Staubli VAL3: movToParkTop.pgx

program movToParkTop()
  local num LnDistance
  local point LpHere
  local point LpPark
begin
  //
  //header begin
  //
  //header end
  //
  stopMove()
  resetMotion()
  // check robot condition:  ESTOP clear, MANUAL MODE, CALIBRATED=true, ARM POWER=ON
  call initializeRobot()
  userPage()
  cls()
  title(" MOVE TO PARK TOP")
  gotoxy(0,4)
  putln("WAITING:  Press MOVE/HOLD button")
  putln("          to move to Park...")
  // put "HALT" in F8 position
  gotoxy(36,13)
  put("HALT")
  //
  //
  bEnableMonitor=true
  LpPark=jointToPoint(tSensorTool,world,jParkTop)
  movel(LpPark,tSensorTool,mGlobalSpeed)
  //
  // watch for Stay Clear Zone entry, process if required
  // watch for bStopMotion initiated from tskHaltMoveMon()
  bWatchForHalt=true
  do
    // get current position, compare with destination
    LpHere=here(tSensorTool,world)
    LpPark=jointToPoint(tSensorTool,world,jPark)
    LnDistance=abs(distance(LpHere,LpPark))
    delay(0)
  until (LnDistance<=nZoneWatchTol) or (bInsideCube==true) or (bInsideCylinder==true) or (bInsideSphere==true) or (bStopMotion==true)
  //
  if (bInsideCube==false) and (bInsideCylinder==false) and (bInsideSphere==false) and (bStopMotion==false)
    waitEndMove()
    popUpMsg("NOW at PARK TOP...Press OK")
  else
    stopMove()
    resetMotion()
    bStopAllMonitor=true
    popUpMsg("MOTION CANCELLED:  Zone Entered or HALT requested; Monitoring Disabled; Manual Recovery REQUIRED...Press OK")
    //
    // put in motion halt recovery steps here
    //
  endIf
  bEnableMonitor=false
  bWatchForHalt=false
  bStopMotion=false
  //
  //
  //done
  //
end
